FUNCTION_BLOCK FB_PropDriveState
VAR_INPUT
	idrive_state 	: INT;
	ipod_state 		: E_PodState;
	bpropFault 		: BOOL;
	propFlag 		: BOOL;
	btimerReset		: BOOL;
END_VAR
VAR_OUTPUT
	btimeOut : BOOL;
END_VAR
VAR
	timerToggle : BOOL;
	fbGracePeriodTimer : TON;
	btrig : BOOL;
END_VAR

timerToggle := FALSE;

IF ((ipod_state <= E_PodState.STATE_HV_ACTIVE OR ipod_state = E_PodState.STATE_MAINTENANCE) AND idrive_state <> 0 AND NOT bPropFault) THEN
	timerToggle := TRUE;
ELSIF ((ipod_state > E_PodState.STATE_HV_ACTIVE AND ipod_state <> E_PodState.STATE_MAINTENANCE) AND idrive_state <> 1 AND NOT bPropFault) THEN
	timerToggle := TRUE;
ELSIF (ipod_state = E_PodState.STATE_MOVEMENT AND propFlag) AND idrive_state <> 2 AND NOT bPropFault THEN
	timerToggle := TRUE;
END_IF
IF NOT btimerReset THEN
	
	fbGracePeriodTimer(IN := timerToggle, PT := T#2S, Q => btrig);

ELSE
	
	fbGracePeriodTimer(IN := FALSE, PT := T#2S);
	btrig := FALSE;
	btimeOut := FALSE;
	
END_IF

IF btrig AND NOT btimerReset THEN
	btimeOut := TRUE;
END_IF

END_FUNCTION_BLOCK

(* stored: Version 1.1.0.1
   POU FB_PropDriveState: Id {7cb0f8de-977c-4fce-a512-5d3a882554fc}, SpecialFunc None *)
